FUNCTION_BLOCK SL_MoveNeedleDown (* MoveNeedleDown: Requires NOT (AtTop AND AtBottom); holds NeedleAxis.Down until (Position >= Distance) OR AtBottom; Invariant NOT (AtTop AND AtBottom) *)
  (* Standard: 61499-2 *)
  (* Version 0.1, 2026-09-28, Project contributors, AAU Smart Production Lab *)
  PACKAGE filler;
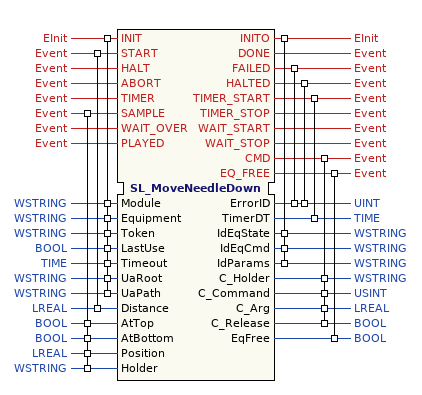
  EVENT_INPUT
    INIT : EInit WITH Module, Equipment, Token, LastUse, Timeout, UaRoot, UaPath;
    START WITH Distance;
    HALT;
    ABORT;
    TIMER;
    SAMPLE WITH AtTop, AtBottom, Position, Holder;
    WAIT_OVER;
    PLAYED;
  END_EVENT
  EVENT_OUTPUT
    INITO : EInit WITH IdEqState, IdEqCmd, IdParams;
    DONE;
    FAILED WITH ErrorID;
    HALTED WITH ErrorID;
    TIMER_START WITH TimerDT;
    TIMER_STOP;
    WAIT_START;
    WAIT_STOP;
    CMD WITH C_Holder, C_Command, C_Arg, C_Release;
    EQ_FREE WITH EqFree;
  END_EVENT
  VAR_INPUT
    Module : WSTRING;
    Equipment : WSTRING;
    Token : WSTRING;
    LastUse : BOOL;
    Timeout : TIME;
    UaRoot : WSTRING;
    UaPath : WSTRING;
    Distance : LREAL;
    AtTop : BOOL;
    AtBottom : BOOL;
    Position : LREAL;
    Holder : WSTRING;
  END_VAR
  VAR_OUTPUT
    ErrorID : UINT;
    TimerDT : TIME;
    IdEqState : WSTRING;
    IdEqCmd : WSTRING;
    IdParams : WSTRING;
    C_Holder : WSTRING;
    C_Command : USINT;
    C_Arg : LREAL;
    C_Release : BOOL;
    EqFree : BOOL;
  END_VAR
  VAR
    Outcome : USINT;
  END_VAR
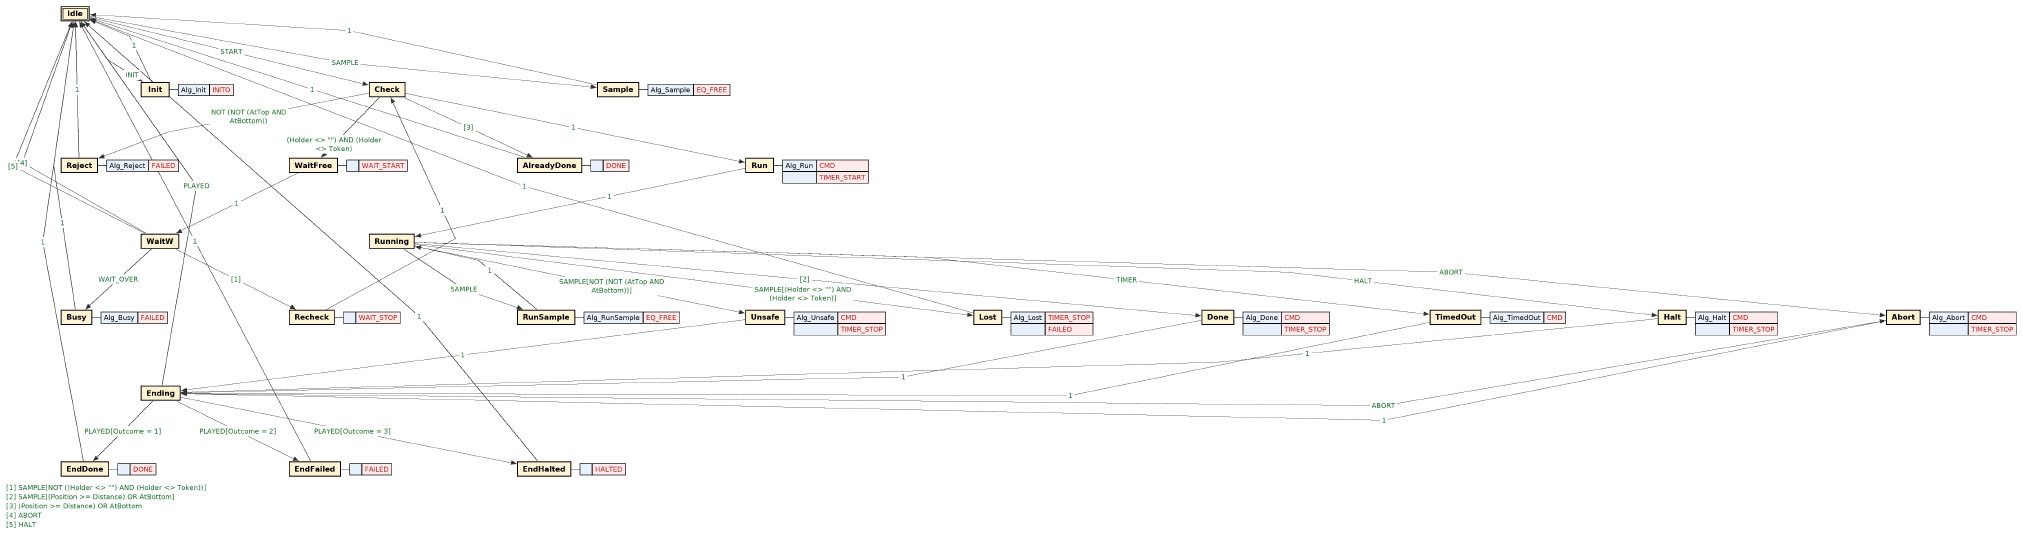
  EC_STATES
    Idle;
    Init : Alg_Init -> INITO;
    Check;
    Reject : Alg_Reject -> FAILED;
    Sample : Alg_Sample -> EQ_FREE;
    Busy : Alg_Busy -> FAILED;
    WaitFree : -> WAIT_START;
    WaitW;
    Recheck : -> WAIT_STOP;
    AlreadyDone : -> DONE;
    Run : Alg_Run -> CMD, -> TIMER_START;
    RunSample : Alg_RunSample -> EQ_FREE;
    Unsafe : Alg_Unsafe -> CMD, -> TIMER_STOP;
    Lost : Alg_Lost -> TIMER_STOP, -> FAILED;
    Done : Alg_Done -> CMD, -> TIMER_STOP;
    TimedOut : Alg_TimedOut -> CMD;
    Halt : Alg_Halt -> CMD, -> TIMER_STOP;
    Abort : Alg_Abort -> CMD, -> TIMER_STOP;
    Ending;
    EndDone : -> DONE;
    EndFailed : -> FAILED;
    EndHalted : -> HALTED;
    Running;
  END_STATES
  EC_TRANSITIONS
    Idle TO Init := INIT;
    Init TO Idle := 1;
    Idle TO Check := START;
    Check TO Reject := NOT (NOT (AtTop AND AtBottom));
    Idle TO Sample := SAMPLE;
    Sample TO Idle := 1;
    Check TO WaitFree := (Holder <> "") AND (Holder <> Token);
    WaitFree TO WaitW := 1;
    WaitW TO Recheck := SAMPLE[NOT ((Holder <> "") AND (Holder <> Token))];
    WaitW TO Busy := WAIT_OVER;
    WaitW TO Idle := HALT;
    WaitW TO Idle := ABORT;
    Recheck TO Check := 1;
    Check TO AlreadyDone := (Position >= Distance) OR AtBottom;
    Running TO Unsafe := SAMPLE[NOT (NOT (AtTop AND AtBottom))];
    Running TO Lost := SAMPLE[(Holder <> "") AND (Holder <> Token)];
    Running TO Done := SAMPLE[(Position >= Distance) OR AtBottom];
    Running TO TimedOut := TIMER;
    Running TO RunSample := SAMPLE;
    RunSample TO Running := 1;
    Busy TO Idle := 1;
    Lost TO Idle := 1;
    AlreadyDone TO Idle := 1;
    Unsafe TO Ending := 1;
    Done TO Ending := 1;
    Halt TO Ending := 1;
    Abort TO Ending := 1;
    TimedOut TO Ending := 1;
    Ending TO EndDone := PLAYED[Outcome = 1];
    Ending TO EndFailed := PLAYED[Outcome = 2];
    Ending TO EndHalted := PLAYED[Outcome = 3];
    Ending TO Idle := PLAYED;
    Ending TO Abort := ABORT;
    EndDone TO Idle := 1;
    EndFailed TO Idle := 1;
    EndHalted TO Idle := 1;
    Check TO Run := 1;
    Run TO Running := 1;
    Running TO Halt := HALT;
    Running TO Abort := ABORT;
    Reject TO Idle := 1;
  END_TRANSITIONS
  ALGORITHM Alg_Init IN ST:
IdEqState := CONCAT(CONCAT(CONCAT(CONCAT("loc[", Module), "/"), Equipment), "/state]");
IdEqCmd := CONCAT(CONCAT(CONCAT(CONCAT("loc[", Module), "/"), Equipment), "/cmd]");
IdParams := CONCAT(CONCAT(CONCAT("opc_ua[WRITE;", CONCAT(UaRoot, UaPath)), "/Parameters/Distance"), "]");
  END_ALGORITHM
  ALGORITHM Alg_Reject IN ST:
ErrorID := 1;
  END_ALGORITHM
  ALGORITHM Alg_Sample IN ST:
EqFree := (Holder = "") OR (Holder = Token);
  END_ALGORITHM
  ALGORITHM Alg_Busy IN ST:
ErrorID := 6;
  END_ALGORITHM
  ALGORITHM Alg_Run IN ST:
C_Holder := Token;
C_Command := 1;
C_Arg := 0.0;
C_Release := FALSE;
TimerDT := Timeout;
  END_ALGORITHM
  ALGORITHM Alg_RunSample IN ST:
EqFree := (Holder = "") OR (Holder = Token);
  END_ALGORITHM
  ALGORITHM Alg_Unsafe IN ST:
C_Holder := Token;
C_Command := 0;
C_Arg := 0.0;
C_Release := LastUse;
ErrorID := 2;
Outcome := 2;
  END_ALGORITHM
  ALGORITHM Alg_Lost IN ST:
ErrorID := 6;
  END_ALGORITHM
  ALGORITHM Alg_Done IN ST:
C_Holder := Token;
C_Command := 0;
C_Arg := 0.0;
C_Release := LastUse;
Outcome := 1;
  END_ALGORITHM
  ALGORITHM Alg_TimedOut IN ST:
C_Holder := Token;
C_Command := 0;
C_Arg := 0.0;
C_Release := LastUse;
ErrorID := 3;
Outcome := 2;
  END_ALGORITHM
  ALGORITHM Alg_Halt IN ST:
C_Holder := Token;
C_Command := 0;
C_Arg := 0.0;
C_Release := LastUse;
ErrorID := 7;
Outcome := 3;
  END_ALGORITHM
  ALGORITHM Alg_Abort IN ST:
C_Holder := Token;
C_Command := 0;
C_Arg := 0.0;
C_Release := TRUE;
Outcome := 0;
  END_ALGORITHM
END_FUNCTION_BLOCK
